PROGRAM P_Demo_FB_HVACPWM
VAR
    fb : FB_HVACPWM;                            // 被演示 FB 实例
    eDataSecurityType_in : E_HVACDataSecurityType ;
    bSetDefault_in : BOOL := FALSE;
    bEnable_in : BOOL := FALSE;
    rYIn_in : REAL := 0.0;
    bReset_in : BOOL := FALSE;
    tPWMPeriod_io : TIME := T#0S;
    tMINPowerOnTime_io : TIME := T#0S;
    bOut_out : BOOL;
    rYOut_out : REAL;
    bInvalidParameter_out : BOOL;
END_VAR

// ============================================================================
// Tc2_HVAC.FB_HVACPWM 演示程序
// ============================================================================
// 场景：把本 FB 实例化到一个 PLC 程序里，每周期单次调用；按需要把 VAR_INPUT 与
//       VAR_IN_OUT 接到工程信号；VAR_OUTPUT 写入对应监视变量。
// 价值：使用本 FB 比手写状态机 / 控制算法节省大量代码；与 Tc2_HVAC 体系内其它 FB
//       直接对接，命名 / 持久化 / 模式仲裁等约定一致。具体语义见 FB_HVACPWM.md 主文档。
// 验证步骤：
//   1. 右键 PLC 项目下 POUs 文件夹 → Add → Existing Item → 选本 .TcPOU 文件
//   2. 引用 Tc2_HVAC（References → Add library）
//   3. 编译 → 登录 → 运行
//   4. 在线写各 *_in 输入信号触发 FB；在线 monitor *_out 引脚观察状态
// ============================================================================

fb(
    eDataSecurityType := eDataSecurityType_in,
    bSetDefault := bSetDefault_in,
    bEnable := bEnable_in,
    rYIn := rYIn_in,
    bReset := bReset_in,
    tPWMPeriod := tPWMPeriod_io,
    tMINPowerOnTime := tMINPowerOnTime_io,
    bOut => bOut_out,
    rYOut => rYOut_out,
    bInvalidParameter => bInvalidParameter_out
);

END_PROGRAM

(* stored: Version 1.1.0.1, ProductVersion 3.1.4024.5
   POU P_Demo_FB_HVACPWM: Id {0efa6bbf-f440-5d53-88b8-7819f5ff9f61}, SpecialFunc None *)
